FUNCTION_BLOCK OR (* Logical OR *)
  (* Standard: 61499-2 *)
  (* Version 1.0, 02.01.2011, gsha041, UoA, Initial Version *)
  (* Compiler header: package fb.rt.UoA; *)
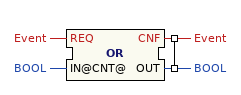
  EVENT_INPUT
    REQ; (* Normal Execution Request *)
  END_EVENT
  EVENT_OUTPUT
    CNF WITH OUT; (* Execution Confirmation *)
  END_EVENT
  VAR_INPUT
    IN@CNT@ : BOOL; (* Argument *)
  END_VAR
  VAR_OUTPUT
    OUT : BOOL; (* Result: IN1 OR IN2 OR ... *)
  END_VAR
END_FUNCTION_BLOCK
